% RSLogix 500 project 9.4.RSS, saved by version 8.30.00.16 %
PROJECT "9.4"    % processor: Bul.1763 MicroLogix 1100 Series B %

PROGRAM FILES
  LAD 2   3 rungs

DATA FILES
  O0 OUTPUT  4 elements
  I1 INPUT  6 elements
  S2 STATUS  66 elements
  B3 BINARY  1 elements
  T4 TIMER  1 elements
  C5 COUNTER  1 elements
  R6 CONTROL  1 elements
  N7 INTEGER  2 elements
  F8 FLOAT  2 elements

LADDER 2
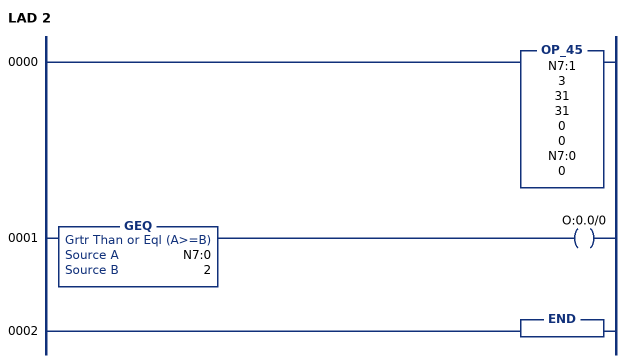
% Rung: 0 %
SOR OP_45 N7:1 3 31 31 0 0 N7:0 0 EOR
% Rung: 1 %
SOR GEQ N7:0 2 OTE O:0.0/0 EOR
% Rung: 2 %
SOR END EOR

DATA TABLE (non-zero values as saved)
DATA N7
% N7:0 % 0 3
DATA F8
% F8:0 % 2 0
